Staubli VAL3: iGrip.pgx

public program iGrip(num& nNum[] (dimensions=1))
begin
  if (dioGet(iGripClosed)==0) and (dioGet(iGripOpen)==1)
    nNum=1
  endIf
  if (dioGet(iGripClosed)==1) and (dioGet(iGripOpen)==0)
    nNum=0
  endIf
end
